FUNCTION_BLOCK FB_3CAM_CameraSequenceNo
VAR_INPUT
	aCameraTrigger		: ARRAY[0..4] OF BOOL;
END_VAR
VAR_OUTPUT

	nCamera1ScanNo		: INT;
	nCamera2ScanNo		: INT;
	nCamera3ScanNo		: INT;
END_VAR
VAR
END_VAR

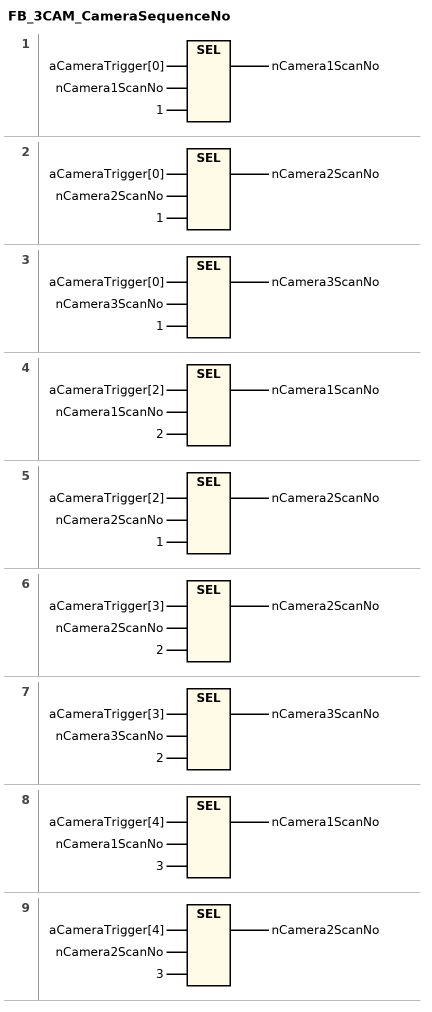
// NETWORK 1
nCamera1ScanNo := SEL(aCameraTrigger[0], nCamera1ScanNo, 1);

// NETWORK 2
nCamera2ScanNo := SEL(aCameraTrigger[0], nCamera2ScanNo, 1);

// NETWORK 3
nCamera3ScanNo := SEL(aCameraTrigger[0], nCamera3ScanNo, 1);

// NETWORK 4
nCamera1ScanNo := SEL(aCameraTrigger[2], nCamera1ScanNo, 2);

// NETWORK 5
nCamera2ScanNo := SEL(aCameraTrigger[2], nCamera2ScanNo, 1);

// NETWORK 6
nCamera2ScanNo := SEL(aCameraTrigger[3], nCamera2ScanNo, 2);

// NETWORK 7
nCamera3ScanNo := SEL(aCameraTrigger[3], nCamera3ScanNo, 2);

// NETWORK 8
nCamera1ScanNo := SEL(aCameraTrigger[4], nCamera1ScanNo, 3);

// NETWORK 9
nCamera2ScanNo := SEL(aCameraTrigger[4], nCamera2ScanNo, 3);

END_FUNCTION_BLOCK

(* stored: Version 1.1.0.1, ProductVersion 3.1.4024.15
   POU FB_3CAM_CameraSequenceNo: Id {eef928a6-4ab3-4c4e-be8b-fb0ce14778e2}, SpecialFunc None *)
